// TIA Portal V19 export
DATA_BLOCK "AUTO_SUBOUTPUT DB"   // DB71
{ S7_Optimized_Access := 'TRUE' }
// stored: MemoryReserve 100
   VAR
      "P-202 A RO 1 FEED PUMP" : Bool;
      "P-202 B RO 1 FEED PUMP" : Bool;
      "P-202 C RO 1 FEED PUMP" : Bool;
      "P-301 A RO 1 HPP PUMP" : Bool;
      "P-301 B RO 1 HPP PUMP" : Bool;
      "P-401 A RO 2 FEED PUMP" : Bool;
      "P-401 B RO 2 FEED PUMP" : Bool;
      "P-401 C RO 2 FEED PUMP" : Bool;
      "P-402  A RO 2 HPP" : Bool;
      "P-402 B" : Bool;
      "P-501 A EDI FEED PUMP" : Bool;
      "P-501 B EDI FEED PUMP" : Bool;
      "P-501 C EDI FEED PUMP" : Bool;
      "EDI 501" : Bool;
      "EDI 502" : Bool;
      "DP 703" : Bool;
      "DP 704" : Bool;
      "DP 705" : Bool;
      "ABV 301" : Bool;
      "ABV 302" : Bool;
      "AGLV-301" : Bool;
      "AGLV-302" : Bool;
      "AGLV-401" : Bool;
      "AGLV-402" : Bool;
      "AGLV-501" : Bool;
      "AGLV-502" : Bool;
   END_VAR
BEGIN
END_DATA_BLOCK
